// Mitsubishi GX Works2 project: LRI   PLC: Q03UDV
// HELLOWORD

// task Task_01 (event TRUE, interval 0, priority 31): POU_01

PROGRAM POU_01
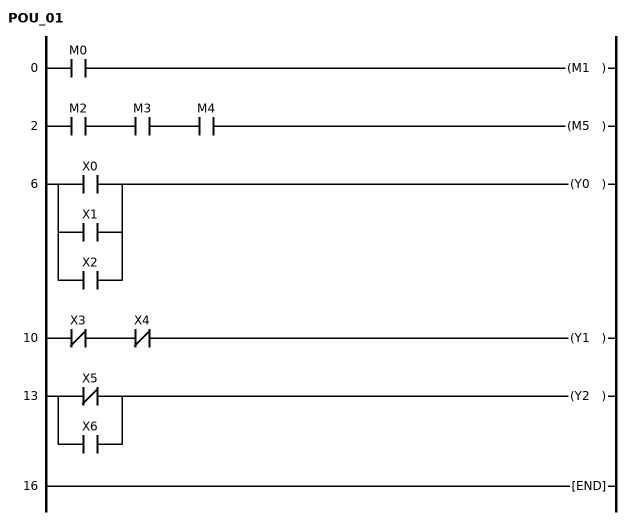
0     LD      M0
      OUT     M1
2     LD      M2
      AND     M3
      AND     M4
      OUT     M5
6     LD      X0
      OR      X1
      OR      X2
      OUT     Y0
10    LDI     X3
      ANI     X4
      OUT     Y1
13    LDI     X5
      OR      X6
      OUT     Y2
16    END
END_PROGRAM
